// TIA Portal V20 export
ORGANIZATION_BLOCK "Main"   // OB1, LAD, ProgramCycle
{ S7_Optimized_Access := 'TRUE' }
VERSION : 0.1
// stored: AutoNumber false, IsIECCheckEnabled false, SetENOAutomatically false
BEGIN

REGION Network 1: 起保停自锁
   // 急停 %I0.2(常闭) 与 停止按钮 %I0.1 串联；启动 %I0.0 与自保持触点 %M0.0 并联后驱动运行标志
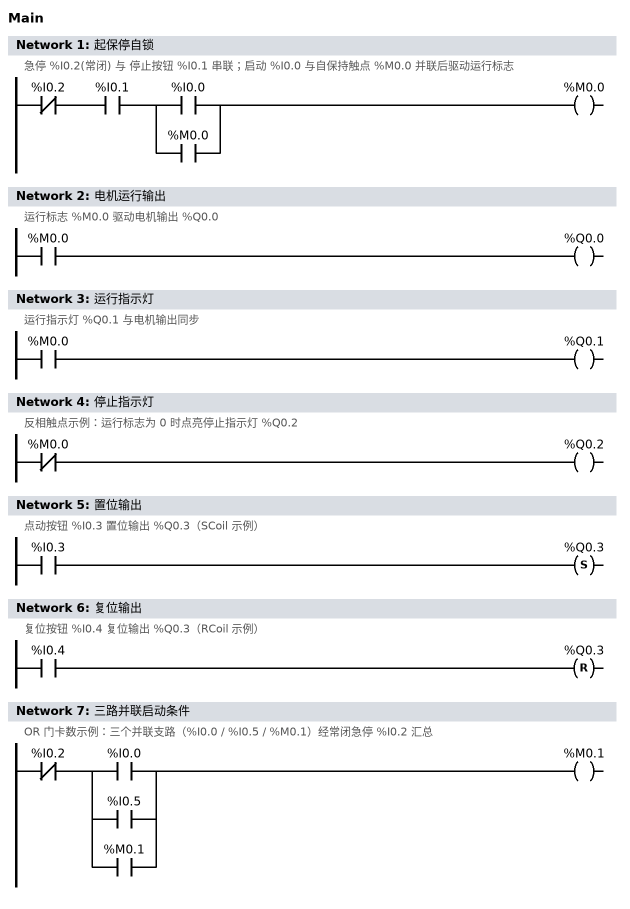
   %M0.0 := NOT %I0.2 AND %I0.1 AND (%I0.0 OR %M0.0);
END_REGION

REGION Network 2: 电机运行输出
   // 运行标志 %M0.0 驱动电机输出 %Q0.0
   RUNG wire#powerrail
      Contact( %M0.0 )
      Coil( %Q0.0 )
   END_RUNG
   // the same network as SCL:
   %Q0.0 := %M0.0;
END_REGION

REGION Network 3: 运行指示灯
   // 运行指示灯 %Q0.1 与电机输出同步
   RUNG wire#powerrail
      Contact( %M0.0 )
      Coil( %Q0.1 )
   END_RUNG
   // the same network as SCL:
   %Q0.1 := %M0.0;
END_REGION

REGION Network 4: 停止指示灯
   // 反相触点示例：运行标志为 0 时点亮停止指示灯 %Q0.2
   RUNG wire#powerrail
      I_Contact( %M0.0 )
      Coil( %Q0.2 )
   END_RUNG
   // the same network as SCL:
   %Q0.2 := NOT %M0.0;
END_REGION

REGION Network 5: 置位输出
   // 点动按钮 %I0.3 置位输出 %Q0.3（SCoil 示例）
   RUNG wire#powerrail
      Contact( %I0.3 )
      S_Coil( %Q0.3 )
   END_RUNG
   // the same network as SCL:
   IF %I0.3 THEN %Q0.3 := TRUE; END_IF;
END_REGION

REGION Network 6: 复位输出
   // 复位按钮 %I0.4 复位输出 %Q0.3（RCoil 示例）
   RUNG wire#powerrail
      Contact( %I0.4 )
      R_Coil( %Q0.3 )
   END_RUNG
   // the same network as SCL:
   IF %I0.4 THEN %Q0.3 := FALSE; END_IF;
END_REGION

REGION Network 7: 三路并联启动条件
   // OR 门卡数示例：三个并联支路（%I0.0 / %I0.5 / %M0.1）经常闭急停 %I0.2 汇总
   %M0.1 := NOT %I0.2 AND (%I0.0 OR %I0.5 OR %M0.1);
END_REGION
END_ORGANIZATION_BLOCK
